SUBAPPLICATION AX_3_3 (* AX_OR and AX_SPLIT for a 3-to-3 Connection *)
  (* Standard: 61499-2 *)
  (* Version 1.0, 2026-09-06, Franz Höpfinger, Meisterschulen am Ostbahnhof, initial API and implementation and/or initial documentation *)
  (* Documentation:
  3 AX-Quellen ODER-verknüpft auf 3 AX-Ziele verteilt
   Kombiniert AX_OR_3 und AX_SPLIT_3 zu einem fertigen Baustein: nimmt IN1/IN2/IN3 entgegen, verknüpft alle drei per ODER zu einem gemeinsamen Signal und verteilt dieses anschließend auf OUT1/OUT2/OUT3.
   Für andere Quellen-/Ziel-Anzahlen: AX_2_2 (2→2), AX_2_3 (2→3), AX_3_2 (3→2).
  *)
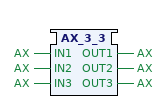
  SOCKETS
    IN1 : adapter::types::unidirectional::AX;
    IN2 : adapter::types::unidirectional::AX;
    IN3 : adapter::types::unidirectional::AX;
  END_SOCKETS
  PLUGS
    OUT1 : adapter::types::unidirectional::AX;
    OUT2 : adapter::types::unidirectional::AX;
    OUT3 : adapter::types::unidirectional::AX;
  END_PLUGS
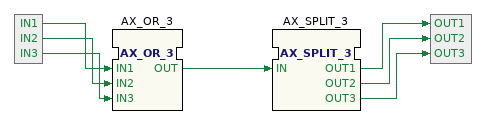
  FBS
    AX_SPLIT_3 : adapter::events::unidirectional::AX_SPLIT_3;
    AX_OR_3 : adapter::booleanOperators::AX_OR_3;
  END_FBS
  ADAPTER_CONNECTIONS
    AX_OR_3.OUT TO AX_SPLIT_3.IN;
    AX_SPLIT_3.OUT1 TO OUT1;
    AX_SPLIT_3.OUT2 TO OUT2;
    AX_SPLIT_3.OUT3 TO OUT3;
    IN1 TO AX_OR_3.IN1;
    IN2 TO AX_OR_3.IN2;
    IN3 TO AX_OR_3.IN3;
  END_CONNECTIONS
END_SUBAPPLICATION
